// TIA Portal project "2020-10-09_Serbatoio" (V16)

(* hardware
DEVICE "S7-1200 station_1"  S7-1200 Station
   slot 0: "Telaio di montaggio_0"  S7-1200 Rack  Rack  V1.0
   slot 1: "PLC_1"  CPU 1215C DC/DC/DC  6ES7 215-1AG40-0XB0  V4.4
*)

// ===== PLC "PLC_1"  CPU 1215C DC/DC/DC =====

VAR_GLOBAL   // PLC tag table "Tabella delle variabili standard"
   "scarico" AT %I0.0 : Bool;
   "s1" AT %I0.1 : Bool;
   "s2" AT %I0.2 : Bool;
   "s3" AT %I0.3 : Bool;
   "s4" AT %I0.4 : Bool;
   "pompa" AT %Q0.0 : Bool;
   "valvola" AT %Q0.1 : Bool;
   "guastoCumulativo" AT %Q0.2 : Bool;
   "guastoS1" AT %M0.0 : Bool;
   "guastoS2" AT %M0.1 : Bool;
   "guastoS3" AT %M0.2 : Bool;
   "guastoS4" AT %M0.3 : Bool;
   "erroreLogica" AT %M0.4 : Bool;
   "ingressi" AT %IB0 : Byte;
   "allarmeSerbatoio" AT %Q0.3 : Bool;
   "ripristinoAllarme" AT %I0.5 : Bool;
END_VAR

// folder: System blocks/Program resources

DATA_BLOCK "TimerSerbatoio"   // DB1
{ S7_Optimized_Access := 'TRUE' }
AUTHOR : Simatic
FAMILY : IEC
NAME : IEC_TMR
VERSION : 1.0
// stored: InstanceOfName IEC_TIMER
"IEC_TIMER"
BEGIN
END_DATA_BLOCK

// folder: (top level)

ORGANIZATION_BLOCK "Main"   // OB1, LAD, ProgramCycle
TITLE = "Main Program Sweep (Cycle)"
{ S7_Optimized_Access := 'TRUE' }
VERSION : 0.1
   VAR_INPUT
      Initial_Call : Bool;   // Initial call of this OB
      Remanence : Bool;   // =True, if remanent data are available
   END_VAR
BEGIN

REGION Network 1: DIAGNOSTICA: guasto cumulativo
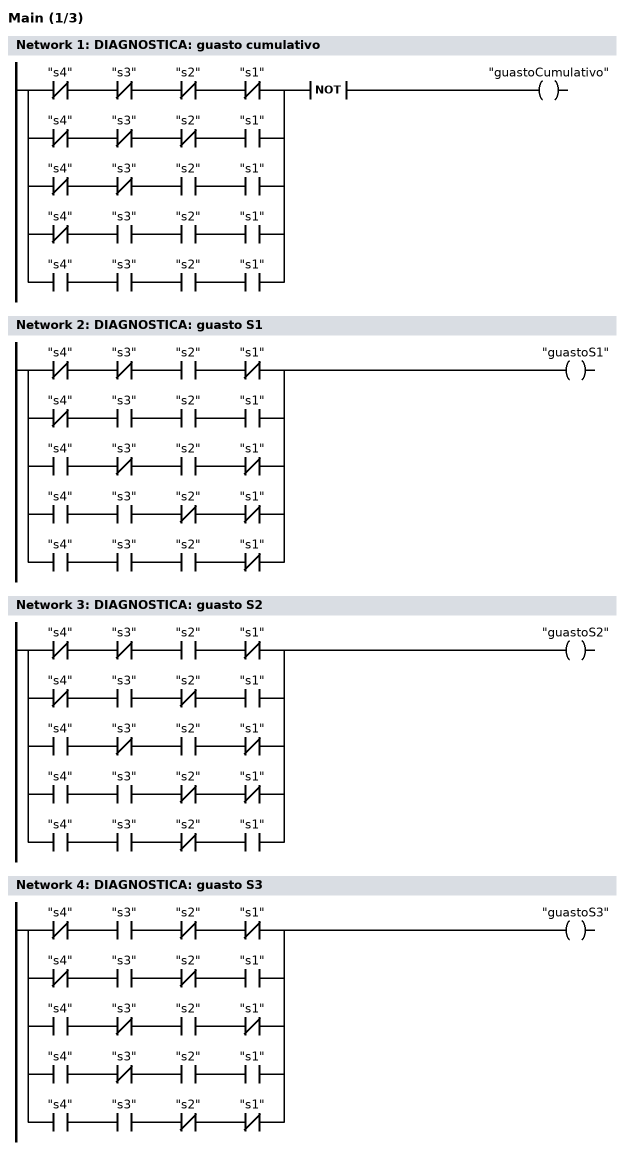
   RUNG wire#powerrail
      I_Contact( "s4" )
      I_Contact( "s3" )
      I_Contact( "s2" )
      I_Contact( "s1" )
      wire#w1
      Not()
      Coil( "guastoCumulativo" )
   END_RUNG
   RUNG wire#powerrail
      I_Contact( "s4" )
      I_Contact( "s3" )
      I_Contact( "s2" )
      Contact( "s1" )
   END_RUNG wire#w1
   RUNG wire#powerrail
      I_Contact( "s4" )
      I_Contact( "s3" )
      Contact( "s2" )
      Contact( "s1" )
   END_RUNG wire#w1
   RUNG wire#powerrail
      I_Contact( "s4" )
      Contact( "s3" )
      Contact( "s2" )
      Contact( "s1" )
   END_RUNG wire#w1
   RUNG wire#powerrail
      Contact( "s4" )
      Contact( "s3" )
      Contact( "s2" )
      Contact( "s1" )
   END_RUNG wire#w1
   // the same network as SCL:
   "guastoCumulativo" := NOT ((NOT "s4" AND NOT "s3" AND NOT "s2" AND NOT "s1") OR (NOT "s4" AND NOT "s3" AND NOT "s2" AND "s1") OR (NOT "s4" AND NOT "s3" AND "s2" AND "s1") OR (NOT "s4" AND "s3" AND "s2" AND "s1") OR ("s4" AND "s3" AND "s2" AND "s1"));
END_REGION

REGION Network 2: DIAGNOSTICA: guasto S1
   RUNG wire#powerrail
      I_Contact( "s4" )
      I_Contact( "s3" )
      Contact( "s2" )
      I_Contact( "s1" )
      wire#w1
      Coil( "guastoS1" )
   END_RUNG
   RUNG wire#powerrail
      I_Contact( "s4" )
      Contact( "s3" )
      Contact( "s2" )
      Contact( "s1" )
   END_RUNG wire#w1
   RUNG wire#powerrail
      Contact( "s4" )
      I_Contact( "s3" )
      Contact( "s2" )
      I_Contact( "s1" )
   END_RUNG wire#w1
   RUNG wire#powerrail
      Contact( "s4" )
      Contact( "s3" )
      I_Contact( "s2" )
      I_Contact( "s1" )
   END_RUNG wire#w1
   RUNG wire#powerrail
      Contact( "s4" )
      Contact( "s3" )
      Contact( "s2" )
      I_Contact( "s1" )
   END_RUNG wire#w1
   // the same network as SCL:
   "guastoS1" := (NOT "s4" AND NOT "s3" AND "s2" AND NOT "s1") OR (NOT "s4" AND "s3" AND "s2" AND "s1") OR ("s4" AND NOT "s3" AND "s2" AND NOT "s1") OR ("s4" AND "s3" AND NOT "s2" AND NOT "s1") OR ("s4" AND "s3" AND "s2" AND NOT "s1");
END_REGION

REGION Network 3: DIAGNOSTICA: guasto S2
   RUNG wire#powerrail
      I_Contact( "s4" )
      I_Contact( "s3" )
      Contact( "s2" )
      I_Contact( "s1" )
      wire#w1
      Coil( "guastoS2" )
   END_RUNG
   RUNG wire#powerrail
      I_Contact( "s4" )
      Contact( "s3" )
      I_Contact( "s2" )
      Contact( "s1" )
   END_RUNG wire#w1
   RUNG wire#powerrail
      Contact( "s4" )
      I_Contact( "s3" )
      Contact( "s2" )
      I_Contact( "s1" )
   END_RUNG wire#w1
   RUNG wire#powerrail
      Contact( "s4" )
      Contact( "s3" )
      I_Contact( "s2" )
      I_Contact( "s1" )
   END_RUNG wire#w1
   RUNG wire#powerrail
      Contact( "s4" )
      Contact( "s3" )
      I_Contact( "s2" )
      Contact( "s1" )
   END_RUNG wire#w1
   // the same network as SCL:
   "guastoS2" := (NOT "s4" AND NOT "s3" AND "s2" AND NOT "s1") OR (NOT "s4" AND "s3" AND NOT "s2" AND "s1") OR ("s4" AND NOT "s3" AND "s2" AND NOT "s1") OR ("s4" AND "s3" AND NOT "s2" AND NOT "s1") OR ("s4" AND "s3" AND NOT "s2" AND "s1");
END_REGION

REGION Network 4: DIAGNOSTICA: guasto S3
   RUNG wire#powerrail
      I_Contact( "s4" )
      Contact( "s3" )
      I_Contact( "s2" )
      I_Contact( "s1" )
      wire#w1
      Coil( "guastoS3" )
   END_RUNG
   RUNG wire#powerrail
      I_Contact( "s4" )
      Contact( "s3" )
      I_Contact( "s2" )
      Contact( "s1" )
   END_RUNG wire#w1
   RUNG wire#powerrail
      Contact( "s4" )
      I_Contact( "s3" )
      Contact( "s2" )
      I_Contact( "s1" )
   END_RUNG wire#w1
   RUNG wire#powerrail
      Contact( "s4" )
      I_Contact( "s3" )
      Contact( "s2" )
      Contact( "s1" )
   END_RUNG wire#w1
   RUNG wire#powerrail
      Contact( "s4" )
      Contact( "s3" )
      I_Contact( "s2" )
      I_Contact( "s1" )
   END_RUNG wire#w1
   // the same network as SCL:
   "guastoS3" := (NOT "s4" AND "s3" AND NOT "s2" AND NOT "s1") OR (NOT "s4" AND "s3" AND NOT "s2" AND "s1") OR ("s4" AND NOT "s3" AND "s2" AND NOT "s1") OR ("s4" AND NOT "s3" AND "s2" AND "s1") OR ("s4" AND "s3" AND NOT "s2" AND NOT "s1");
END_REGION

REGION Network 5: DIAGNOSTICA: guasto S4
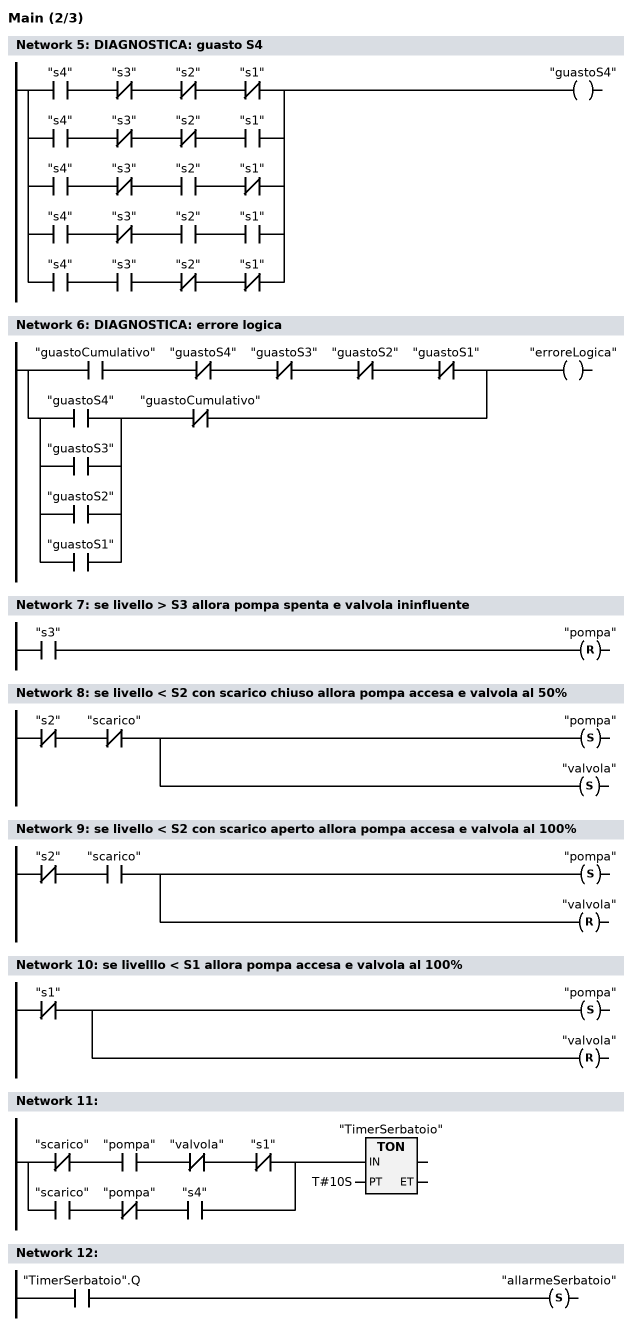
   RUNG wire#powerrail
      Contact( "s4" )
      I_Contact( "s3" )
      I_Contact( "s2" )
      I_Contact( "s1" )
      wire#w1
      Coil( "guastoS4" )
   END_RUNG
   RUNG wire#powerrail
      Contact( "s4" )
      I_Contact( "s3" )
      I_Contact( "s2" )
      Contact( "s1" )
   END_RUNG wire#w1
   RUNG wire#powerrail
      Contact( "s4" )
      I_Contact( "s3" )
      Contact( "s2" )
      I_Contact( "s1" )
   END_RUNG wire#w1
   RUNG wire#powerrail
      Contact( "s4" )
      I_Contact( "s3" )
      Contact( "s2" )
      Contact( "s1" )
   END_RUNG wire#w1
   RUNG wire#powerrail
      Contact( "s4" )
      Contact( "s3" )
      I_Contact( "s2" )
      I_Contact( "s1" )
   END_RUNG wire#w1
   // the same network as SCL:
   "guastoS4" := ("s4" AND NOT "s3" AND NOT "s2" AND NOT "s1") OR ("s4" AND NOT "s3" AND NOT "s2" AND "s1") OR ("s4" AND NOT "s3" AND "s2" AND NOT "s1") OR ("s4" AND NOT "s3" AND "s2" AND "s1") OR ("s4" AND "s3" AND NOT "s2" AND NOT "s1");
END_REGION

REGION Network 6: DIAGNOSTICA: errore logica
   RUNG wire#powerrail
      Contact( "guastoCumulativo" )
      I_Contact( "guastoS4" )
      I_Contact( "guastoS3" )
      I_Contact( "guastoS2" )
      I_Contact( "guastoS1" )
      wire#w1
      Coil( "erroreLogica" )
   END_RUNG
   RUNG wire#powerrail
      Contact( "guastoS4" )
      wire#w2
      I_Contact( "guastoCumulativo" )
   END_RUNG wire#w1
   RUNG wire#powerrail
      Contact( "guastoS3" )
   END_RUNG wire#w2
   RUNG wire#powerrail
      Contact( "guastoS2" )
   END_RUNG wire#w2
   RUNG wire#powerrail
      Contact( "guastoS1" )
   END_RUNG wire#w2
   // the same network as SCL:
   "erroreLogica" := ("guastoCumulativo" AND NOT "guastoS4" AND NOT "guastoS3" AND NOT "guastoS2" AND NOT "guastoS1") OR (("guastoS4" OR "guastoS3" OR "guastoS2" OR "guastoS1") AND NOT "guastoCumulativo");
END_REGION

REGION Network 7: se livello > S3 allora pompa spenta e valvola ininfluente
   RUNG wire#powerrail
      Contact( "s3" )
      R_Coil( "pompa" )
   END_RUNG
   // the same network as SCL:
   IF "s3" THEN "pompa" := FALSE; END_IF;
END_REGION

REGION Network 8: se livello < S2 con scarico chiuso allora pompa accesa e valvola al 50%
   RUNG wire#powerrail
      I_Contact( "s2" )
      I_Contact( "scarico" )
      wire#w1
      S_Coil( "pompa" )
   END_RUNG
   RUNG wire#w1
      S_Coil( "valvola" )
   END_RUNG
   // the same network as SCL:
   IF NOT "s2" AND NOT "scarico" THEN
       "pompa" := TRUE;
       "valvola" := TRUE;
   END_IF;
END_REGION

REGION Network 9: se livello < S2 con scarico aperto allora pompa accesa e valvola al 100%
   RUNG wire#powerrail
      I_Contact( "s2" )
      Contact( "scarico" )
      wire#w1
      S_Coil( "pompa" )
   END_RUNG
   RUNG wire#w1
      R_Coil( "valvola" )
   END_RUNG
   // the same network as SCL:
   IF NOT "s2" AND "scarico" THEN
       "pompa" := TRUE;
       "valvola" := FALSE;
   END_IF;
END_REGION

REGION Network 10: se livelllo < S1 allora pompa accesa e valvola al 100%
   RUNG wire#powerrail
      I_Contact( "s1" )
      wire#w1
      S_Coil( "pompa" )
   END_RUNG
   RUNG wire#w1
      R_Coil( "valvola" )
   END_RUNG
   // the same network as SCL:
   IF NOT "s1" THEN
       "pompa" := TRUE;
       "valvola" := FALSE;
   END_IF;
END_REGION

REGION Network 11
   "TimerSerbatoio".TON(IN := (NOT "scarico" AND "pompa" AND NOT "valvola" AND NOT "s1") OR ("scarico" AND NOT "pompa" AND "s4"),
                        PT := T#10S);
END_REGION

REGION Network 12
   RUNG wire#powerrail
      Contact( "TimerSerbatoio".Q )
      S_Coil( "allarmeSerbatoio" )
   END_RUNG
   // the same network as SCL:
   IF "TimerSerbatoio".Q THEN "allarmeSerbatoio" := TRUE; END_IF;
END_REGION

REGION Network 13
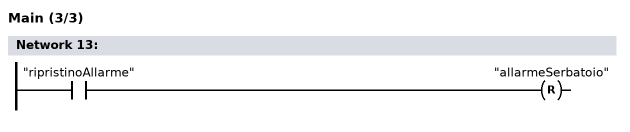
   RUNG wire#powerrail
      Contact( "ripristinoAllarme" )
      R_Coil( "allarmeSerbatoio" )
   END_RUNG
   // the same network as SCL:
   IF "ripristinoAllarme" THEN "allarmeSerbatoio" := FALSE; END_IF;
END_REGION
END_ORGANIZATION_BLOCK